SUBAPPLICATION GreenWhiteBackground4C (* Hintergrundfarbe (TRUE -> Grün, FALSE -> Weiß) für 4 Objekte (Kompakt) *)
  (* Standard: 61499-2 *)
  (* Version 1.0, 2023-02-11, franz, Meisterschulen am Ostbahnhof *)
  PACKAGE MyLib::sys;
  IMPORT isobus::UT::Q::const::IDs::ID_NULL;
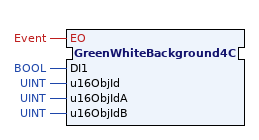
  EVENT_INPUT
    EO;
  END_EVENT
  VAR_INPUT
    DI1 : BOOL; (* Selector *)
    u16ObjId : UINT := ID_NULL; (* Object ID Softkey *)
    u16ObjIdA : UINT := ID_NULL; (* Object ID AUX *)
    u16ObjIdB : UINT := ID_NULL; (* Object ID Button *)
  END_VAR
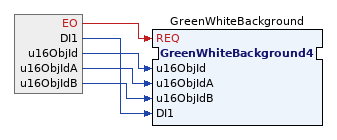
  SUBAPPS
    GreenWhiteBackground : MyLib::sys::GreenWhiteBackground4;
  END_SUBAPPS
  EVENT_CONNECTIONS
    EO TO GreenWhiteBackground.REQ;
  END_CONNECTIONS
  DATA_CONNECTIONS
    u16ObjId TO GreenWhiteBackground.u16ObjId;
    u16ObjIdA TO GreenWhiteBackground.u16ObjIdA;
    u16ObjIdB TO GreenWhiteBackground.u16ObjIdB;
    DI1 TO GreenWhiteBackground.DI1;
  END_CONNECTIONS
END_SUBAPPLICATION
